{attribute 'qualified_only'}
{attribute 'strict'}
TYPE EAssertion_t :
(
	eStatePassed,
	eStateFailed,
	eStateFailedFatal
);
END_TYPE

(* stored: Version 1.1.0.1, ProductVersion 3.1.4024.11
   DUT EAssertion_t: Id {718fcced-2366-499d-bde0-c52581db0fd1} *)
